PROGRAM Tests
VAR
	eventHandlers_Test : EventHandlers_Test;
END_VAR

eventHandlers_Test();

END_PROGRAM

(* stored: Version 1.1.0.1, ProductVersion 3.1.4024.12
   POU Tests: Id {716cf7d2-4a71-4aac-8d46-2dbbbbf0001b}, SpecialFunc None *)
